FUNCTION_BLOCK FB_Sample_07_MeasurementDataChannel
VAR_INPUT
	nStateChannel		AT%I*	: USINT;
	nScale				AT%I*	: SINT;
	MVDistance			AT%I*	: INT;
END_VAR
VAR_OUTPUT
	bValid						: BOOL;
	bError						: BOOL;
	nValueStatus				: E_IolMdc_ValueStatus;
	nValueDINT					: DINT;
	nValueREAL					: LREAL;
	nScaleOut					: INT;
END_VAR
VAR
	fbMeasurement				: IOL_MeasurementDataChannel_INT;
END_VAR

fbMeasurement
(
	Enable := TRUE, 
	SubstituteValue := 500, 
	ChannelState := nStateChannel, 
	ScaleIn := nScale, 
	MeasurementValue := MVDistance, 
	Valid => bValid, 
	Error => bError, 
	ValueStatus => nValueStatus, 
	ValueReal => nValueREAL, 
	ValueDINT => nValueDINT, 
	Scale => nScaleOut 
);

END_FUNCTION_BLOCK

(* stored: Version 1.1.0.1, ProductVersion 3.1.4024.11
   POU FB_Sample_07_MeasurementDataChannel: Id {ff115613-3ab5-49e8-95be-58e038c26551}, SpecialFunc None *)
